// sample about how to export filtered logged events
PROGRAM Sample_ExportFilter
VAR
	hr : HRESULT;
	
	bExport				: BOOL;
	fbCsvExportSetting	: FB_TcEventCsvExportSettings; 
	fbExportFilter		: FB_TcEventFilter; 
	sExportFileName		: STRING := 'c:\temp\Eventlogger-export.csv';
	
	fbEventLogger	: FB_TcEventLogger;
	fbTrig			: R_TRIG;
END_VAR

//this exports the messages with 'MessageTest' eventclass but not the alarms
fbTrig(CLK:=bExport);
IF bExport THEN
	IF fbTrig.Q THEN 
		fbCsvExportSetting.Clear();
		fbCsvExportSetting.AddLanguage(TcLcid.de_DE, 'German');
		fbCsvExportSetting.AddFilter(fbExportFilter); 
		fbExportFilter.Clear().IsMessage().AND_OP().EventClass.EqualTo(TC_EVENTS.MessageTest.Message.uuidEventClass);
	END_IF
	bExport := NOT fbEventLogger.ExportLoggedEvents(sExportFileName, fbCsvExportSetting, hrErrorCode=>hr);// async request returns TRUE if not any more busy 
END_IF

END_PROGRAM

(* stored: Version 1.1.0.1, ProductVersion 3.1.4024.12
   POU Sample_ExportFilter: Id {22d7733b-ca62-4e25-bc67-09ac3bdc7973}, SpecialFunc None *)
